{attribute 'qualified_only'}
{attribute 'strict'}
{attribute 'to_string'}
TYPE eSchuifStates :
(
	enum_member := 0
);
END_TYPE

(* stored: Version 1.1.0.1
   DUT eSchuifStates: Id {9bdae2b2-7b86-42b0-8ece-b2c3a4e72d8f} *)
